Yaskawa INFORM job: ARGAZ5.JBI

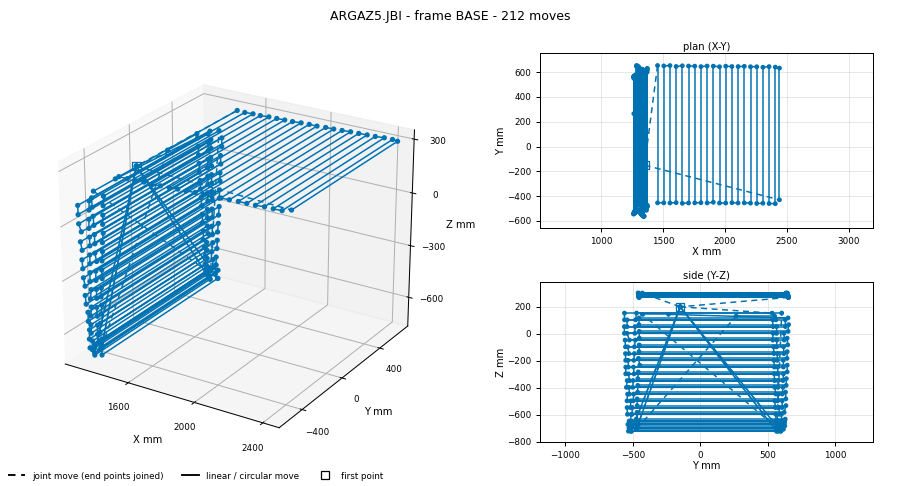
[picture p0: tool path of ARGAZ5.JBI in frame BASE, 212 of 212 moves have a stored position in this frame; points joined in program order, loops and branches not executed]
/JOB
//NAME ARGAZ5
//POS
///NPOS 206,0,206,1,0,1
///TOOL 0
///POSTYPE BASE
///RECTAN
///RCONF 0,0,0,0,0,0,0,0,0,0,0,0,0,0,0,0,0,0,0,0,0,0,0,0
C00000=2438.372,-429.843,302.316,175.0000,5.0000,175.0000
C00001=2438.372,633.343,302.316,175.0000,5.0000,175.0000
C00002=2404.704,640.901,302.803,175.0000,5.0000,175.0000
C00003=2404.704,-461.113,302.803,175.0000,5.0000,175.0000
C00004=2354.704,-459.538,300.563,175.0000,5.0000,175.0000
C00005=2354.704,645.007,300.563,175.0000,5.0000,175.0000
C00006=2304.704,639.966,299.253,175.0000,5.0000,175.0000
C00007=2304.704,-457.215,299.253,175.0000,5.0000,175.0000
C00008=2254.704,-459.172,296.365,175.0000,5.0000,175.0000
C00009=2254.704,644.031,296.365,175.0000,5.0000,175.0000
C00010=2204.704,644.248,294.144,175.0000,5.0000,175.0000
C00011=2204.704,-456.654,294.144,175.0000,5.0000,175.0000
C00012=2154.704,-454.150,292.149,175.0000,5.0000,175.0000
C00013=2154.704,647.282,292.149,175.0000,5.0000,175.0000
C00014=2104.704,645.426,290.068,175.0000,5.0000,175.0000
C00015=2104.704,-455.328,290.068,175.0000,5.0000,175.0000
C00016=2054.704,-453.054,287.793,175.0000,5.0000,175.0000
C00017=2054.704,645.839,287.793,175.0000,5.0000,175.0000
C00018=2004.704,648.293,285.625,175.0000,5.0000,175.0000
C00019=2004.704,-455.974,285.625,175.0000,5.0000,175.0000
C00020=1954.704,-455.663,284.513,175.0000,5.0000,175.0000
C00021=1954.704,644.044,284.513,175.0000,5.0000,175.0000
C00022=1904.704,648.760,282.533,175.0000,5.0000,175.0000
C00023=1904.704,-449.454,282.533,175.0000,5.0000,175.0000
C00024=1854.704,-454.861,280.617,175.0000,5.0000,175.0000
C00025=1854.704,649.609,280.617,175.0000,5.0000,175.0000
C00026=1804.704,645.165,279.272,175.0000,5.0000,175.0000
C00027=1804.704,-453.058,279.272,175.0000,5.0000,175.0000
C00028=1754.704,-454.350,276.998,175.0000,5.0000,175.0000
C00029=1754.704,648.797,276.998,175.0000,5.0000,175.0000
C00030=1704.704,649.851,275.425,175.0000,5.0000,175.0000
C00031=1704.704,-455.236,275.425,175.0000,5.0000,175.0000
C00032=1654.704,-457.856,273.661,175.0000,5.0000,175.0000
C00033=1654.704,651.982,273.661,175.0000,5.0000,175.0000
C00034=1604.704,646.210,272.661,175.0000,5.0000,175.0000
C00035=1604.704,-452.258,272.661,175.0000,5.0000,175.0000
C00036=1554.704,-455.193,270.474,175.0000,5.0000,175.0000
C00037=1554.704,653.496,270.474,175.0000,5.0000,175.0000
C00038=1504.704,650.879,269.338,175.0000,5.0000,175.0000
C00039=1504.704,-454.045,269.338,175.0000,5.0000,175.0000
C00040=1454.676,-454.040,269.843,175.0000,5.0000,175.0000
C00041=1454.676,653.895,269.843,175.0000,5.0000,175.0000
C00042=1347.088,531.287,153.366,175.0000,-89.9999,5.0000
C00043=1347.088,-562.394,153.366,175.0000,-89.9999,5.0000
C00044=1344.164,-562.287,103.366,175.0000,-89.9999,5.0000
C00045=1344.164,534.938,103.366,175.0000,-89.9999,5.0000
C00046=1342.438,538.625,53.366,175.0000,-89.9999,5.0000
C00047=1342.438,-562.994,53.366,175.0000,-89.9999,5.0000
C00048=1340.832,-563.178,3.366,175.0000,-89.9999,5.0000
C00049=1340.832,538.871,3.366,175.0000,-89.9999,5.0000
C00050=1338.825,536.219,-46.633,175.0000,-89.9999,5.0000
C00051=1338.825,-558.107,-46.633,175.0000,-89.9999,5.0000
C00052=1337.044,-554.870,-96.633,175.0000,-89.9999,5.0000
C00053=1337.044,542.164,-96.633,175.0000,-89.9999,5.0000
C00054=1335.183,545.111,-146.633,175.0000,-89.9999,5.0000
C00055=1335.183,-555.018,-146.633,175.0000,-89.9999,5.0000
C00056=1333.293,-553.493,-196.633,175.0000,-89.9999,5.0000
C00057=1333.293,545.184,-196.633,175.0000,-89.9999,5.0000
C00058=1331.807,548.689,-246.633,175.0000,-89.9999,5.0000
C00059=1331.807,-552.923,-246.633,175.0000,-89.9999,5.0000
C00060=1329.870,-553.256,-296.633,175.0000,-89.9999,5.0000
C00061=1329.870,547.209,-296.633,175.0000,-89.9999,5.0000
C00062=1327.995,549.873,-346.633,175.0000,-89.9999,5.0000
C00063=1327.995,-542.334,-346.633,175.0000,-89.9999,5.0000
C00064=1326.213,-548.248,-396.633,175.0000,-89.9999,5.0000
C00065=1326.213,550.626,-396.633,175.0000,-89.9999,5.0000
C00066=1324.396,560.131,-446.633,175.0000,-89.9999,5.0000
C00067=1324.396,-539.231,-446.633,175.0000,-89.9999,5.0000
C00068=1322.129,-543.451,-496.633,175.0000,-89.9999,5.0000
C00069=1322.129,550.722,-496.633,175.0000,-89.9999,5.0000
C00070=1320.170,556.350,-546.633,175.0000,-89.9999,5.0000
C00071=1320.170,-543.270,-546.633,175.0000,-89.9999,5.0000
C00072=1318.250,-540.170,-596.633,175.0000,-89.9999,5.0000
C00073=1318.250,558.973,-596.633,175.0000,-89.9999,5.0000
C00074=1316.642,560.301,-646.633,175.0000,-89.9999,5.0000
C00075=1316.642,-527.964,-646.633,175.0000,-89.9999,5.0000
C00076=1314.806,-529.352,-696.633,175.0000,-89.9999,5.0000
C00077=1314.806,561.085,-696.633,175.0000,-89.9999,5.0000
C00078=1333.412,565.195,-671.633,180.0000,-60.0000,0.0000
C00079=1333.412,-537.251,-671.633,180.0000,-60.0000,0.0000
C00080=1332.156,-533.079,-721.633,180.0000,-60.0000,0.0000
C00081=1332.156,565.345,-721.633,180.0000,-60.0000,0.0000
C00082=1332.156,565.345,-721.633,180.0000,-60.0000,0.0000
C00083=1371.377,602.641,153.649,175.0000,-89.9999,5.0000
C00084=1371.377,-472.613,153.649,175.0000,-89.9999,5.0000
C00085=1372.180,-480.408,103.649,175.0000,-89.9999,5.0000
C00086=1372.180,629.123,103.649,175.0000,-89.9999,5.0000
C00087=1371.089,629.796,53.649,175.0000,-89.9999,5.0000
C00088=1371.089,-483.667,53.649,175.0000,-89.9999,5.0000
C00089=1369.998,-485.573,3.649,175.0000,-89.9999,5.0000
C00090=1369.998,619.394,3.649,175.0000,-89.9999,5.0000
C00091=1369.110,621.830,-46.350,175.0000,-89.9999,5.0000
C00092=1369.110,-481.873,-46.350,175.0000,-89.9999,5.0000
C00093=1367.639,-488.976,-96.350,175.0000,-89.9999,5.0000
C00094=1367.639,616.630,-96.350,175.0000,-89.9999,5.0000
C00095=1366.582,618.500,-146.350,175.0000,-89.9999,5.0000
C00096=1366.582,-488.746,-146.350,175.0000,-89.9999,5.0000
C00097=1365.085,-493.213,-196.350,175.0000,-89.9999,5.0000
C00098=1365.085,614.650,-196.350,175.0000,-89.9999,5.0000
C00099=1363.658,614.990,-246.350,175.0000,-89.9999,5.0000
C00100=1363.658,-495.754,-246.350,175.0000,-89.9999,5.0000
C00101=1361.864,-491.909,-296.350,175.0000,-89.9999,5.0000
C00102=1361.864,615.571,-296.350,175.0000,-89.9999,5.0000
C00103=1360.073,611.872,-346.350,175.0000,-89.9999,5.0000
C00104=1360.073,-498.655,-346.350,175.0000,-89.9999,5.0000
C00105=1358.161,-500.748,-396.350,175.0000,-89.9999,5.0000
C00106=1358.161,611.928,-396.350,175.0000,-89.9999,5.0000
C00107=1356.405,607.009,-446.350,175.0000,-89.9999,5.0000
C00108=1356.405,-493.709,-446.350,175.0000,-89.9999,5.0000
C00109=1354.608,-498.341,-496.350,175.0000,-89.9999,5.0000
C00110=1354.608,606.376,-496.350,175.0000,-89.9999,5.0000
C00111=1352.468,605.807,-546.350,175.0000,-89.9999,5.0000
C00112=1352.468,-503.981,-546.350,175.0000,-89.9999,5.0000
C00113=1350.405,-507.600,-596.350,175.0000,-89.9999,5.0000
C00114=1350.405,600.519,-596.350,175.0000,-89.9999,5.0000
C00115=1348.479,602.258,-646.350,175.0000,-89.9999,5.0000
C00116=1348.479,-507.412,-646.350,175.0000,-89.9999,5.0000
C00117=1346.462,-509.588,-696.350,175.0000,-89.9999,5.0000
C00118=1346.462,597.739,-696.350,175.0000,-89.9999,5.0000
C00119=1364.869,596.218,-671.350,180.0000,-60.0000,0.0000
C00120=1364.869,-512.867,-671.350,180.0000,-60.0000,0.0000
C00121=1363.104,-512.908,-721.350,180.0000,-60.0000,0.0000
C00122=1363.104,596.344,-721.350,180.0000,-60.0000,0.0000
C00123=1363.104,596.344,-721.350,180.0000,-60.0000,0.0000
C00124=1277.888,-429.618,144.199,175.0000,-89.9999,5.0000
C00125=1277.888,-236.558,144.199,175.0000,-89.9999,5.0000
C00126=1283.410,649.398,117.816,175.0000,-89.9999,5.0000
C00127=1283.410,-454.812,117.816,175.0000,-89.9999,5.0000
C00128=1286.253,-455.480,67.816,175.0000,-89.9999,5.0000
C00129=1286.253,653.737,67.816,175.0000,-89.9999,5.0000
C00130=1288.733,650.101,17.816,175.0000,-89.9999,5.0000
C00131=1288.733,-453.231,17.816,175.0000,-89.9999,5.0000
C00132=1291.050,-452.345,-32.183,175.0000,-89.9999,5.0000
C00133=1291.050,643.233,-32.183,175.0000,-89.9999,5.0000
C00134=1293.592,647.319,-82.183,175.0000,-89.9999,5.0000
C00135=1293.592,-453.386,-82.183,175.0000,-89.9999,5.0000
C00136=1295.614,-454.881,-132.183,175.0000,-89.9999,5.0000
C00137=1295.614,643.520,-132.183,175.0000,-89.9999,5.0000
C00138=1297.247,642.008,-182.183,175.0000,-89.9999,5.0000
C00139=1297.247,-459.228,-182.183,175.0000,-89.9999,5.0000
C00140=1299.433,-449.216,-232.183,175.0000,-89.9999,5.0000
C00141=1299.433,643.471,-232.183,175.0000,-89.9999,5.0000
C00142=1300.418,643.420,-282.183,175.0000,-89.9999,5.0000
C00143=1300.418,-460.256,-282.183,175.0000,-89.9999,5.0000
C00144=1302.234,-463.734,-332.183,175.0000,-89.9999,5.0000
C00145=1302.234,636.925,-332.183,175.0000,-89.9999,5.0000
C00146=1303.707,635.868,-382.183,175.0000,-89.9999,5.0000
C00147=1303.707,-463.869,-382.183,175.0000,-89.9999,5.0000
C00148=1305.086,-465.019,-432.183,175.0000,-89.9999,5.0000
C00149=1305.086,630.756,-432.183,175.0000,-89.9999,5.0000
C00150=1306.071,633.429,-482.183,175.0000,-89.9999,5.0000
C00151=1306.071,-468.802,-482.183,175.0000,-89.9999,5.0000
C00152=1307.412,-468.117,-532.183,175.0000,-89.9999,5.0000
C00153=1307.412,633.875,-532.183,175.0000,-89.9999,5.0000
C00154=1308.466,621.089,-582.183,175.0000,-89.9999,5.0000
C00155=1308.466,-469.996,-582.183,175.0000,-89.9999,5.0000
C00156=1310.304,-475.204,-632.183,175.0000,-89.9999,5.0000
C00157=1310.304,628.888,-632.183,175.0000,-89.9999,5.0000
C00158=1311.312,625.813,-682.183,175.0000,-89.9999,5.0000
C00159=1311.312,-473.494,-682.183,175.0000,-89.9999,5.0000
C00160=1332.658,-465.818,-657.183,180.0000,-60.0000,0.0000
C00161=1332.658,624.168,-657.183,180.0000,-60.0000,0.0000
C00162=1333.118,615.110,-707.183,180.0000,-60.0000,0.0000
C00163=1333.118,-474.618,-707.183,180.0000,-60.0000,0.0000
C00164=1333.118,-474.618,-707.183,180.0000,-60.0000,0.0000
C00165=1263.288,265.502,131.277,175.0000,-89.9999,5.0000
C00166=1263.288,550.035,131.277,175.0000,-89.9999,5.0000
C00167=1260.890,559.755,103.296,175.0000,-89.9999,5.0000
C00168=1260.890,-543.266,103.296,175.0000,-89.9999,5.0000
C00169=1261.533,-543.209,53.296,175.0000,-89.9999,5.0000
C00170=1261.533,565.502,53.296,175.0000,-89.9999,5.0000
C00171=1263.366,564.257,3.296,175.0000,-89.9999,5.0000
C00172=1263.366,-543.096,3.296,175.0000,-89.9999,5.0000
C00173=1265.404,-525.948,-46.703,175.0000,-89.9999,5.0000
C00174=1265.404,566.502,-46.703,175.0000,-89.9999,5.0000
C00175=1267.028,564.815,-96.703,175.0000,-89.9999,5.0000
C00176=1267.028,-538.386,-96.703,175.0000,-89.9999,5.0000
C00177=1269.183,-528.977,-146.703,175.0000,-89.9999,5.0000
C00178=1269.183,570.662,-146.703,175.0000,-89.9999,5.0000
C00179=1270.966,569.787,-196.703,175.0000,-89.9999,5.0000
C00180=1270.966,-535.503,-196.703,175.0000,-89.9999,5.0000
C00181=1272.925,-533.396,-246.703,175.0000,-89.9999,5.0000
C00182=1272.925,572.645,-246.703,175.0000,-89.9999,5.0000
C00183=1275.047,573.565,-296.703,175.0000,-89.9999,5.0000
C00184=1275.047,-533.499,-296.703,175.0000,-89.9999,5.0000
C00185=1277.369,-524.427,-346.703,175.0000,-89.9999,5.0000
C00186=1277.369,576.345,-346.703,175.0000,-89.9999,5.0000
C00187=1279.521,573.757,-396.703,175.0000,-89.9999,5.0000
C00188=1279.521,-528.930,-396.703,175.0000,-89.9999,5.0000
C00189=1281.635,-525.764,-446.703,175.0000,-89.9999,5.0000
C00190=1281.635,579.175,-446.703,175.0000,-89.9999,5.0000
C00191=1283.849,571.736,-496.703,175.0000,-89.9999,5.0000
C00192=1283.849,-515.793,-496.703,175.0000,-89.9999,5.0000
C00193=1285.977,-517.912,-546.703,175.0000,-89.9999,5.0000
C00194=1285.977,582.744,-546.703,175.0000,-89.9999,5.0000
C00195=1288.303,585.349,-596.703,175.0000,-89.9999,5.0000
C00196=1288.303,-512.618,-596.703,175.0000,-89.9999,5.0000
C00197=1290.270,-519.107,-646.703,175.0000,-89.9999,5.0000
C00198=1290.270,579.567,-646.703,175.0000,-89.9999,5.0000
C00199=1292.656,581.655,-696.703,175.0000,-89.9999,5.0000
C00200=1292.656,-518.761,-696.703,175.0000,-89.9999,5.0000
C00201=1314.870,-511.376,-671.703,180.0000,-60.0000,0.0000
C00202=1314.870,581.349,-671.703,180.0000,-60.0000,0.0000
C00203=1317.105,581.261,-721.703,180.0000,-60.0000,0.0000
C00204=1317.105,-511.969,-721.703,180.0000,-60.0000,0.0000
C00205=1317.105,-511.969,-721.703,180.0000,-60.0000,0.0000
///POSTYPE PULSE
///PULSE
EC00000=0
EC00001=0
EC00002=0
EC00003=0
EC00004=0
EC00005=0
EC00006=0
EC00007=0
EC00008=0
EC00009=0
EC00010=0
EC00011=0
EC00012=0
EC00013=0
EC00014=0
EC00015=0
EC00016=0
EC00017=0
EC00018=0
EC00019=0
EC00020=0
EC00021=0
EC00022=0
EC00023=0
EC00024=0
EC00025=0
EC00026=0
EC00027=0
EC00028=0
EC00029=0
EC00030=0
EC00031=0
EC00032=0
EC00033=0
EC00034=0
EC00035=0
EC00036=0
EC00037=0
EC00038=0
EC00039=0
EC00040=0
EC00041=0
EC00042=0
EC00043=0
EC00044=0
EC00045=0
EC00046=0
EC00047=0
EC00048=0
EC00049=0
EC00050=0
EC00051=0
EC00052=0
EC00053=0
EC00054=0
EC00055=0
EC00056=0
EC00057=0
EC00058=0
EC00059=0
EC00060=0
EC00061=0
EC00062=0
EC00063=0
EC00064=0
EC00065=0
EC00066=0
EC00067=0
EC00068=0
EC00069=0
EC00070=0
EC00071=0
EC00072=0
EC00073=0
EC00074=0
EC00075=0
EC00076=0
EC00077=0
EC00078=0
EC00079=0
EC00080=0
EC00081=0
EC00082=92160
EC00083=92160
EC00084=92160
EC00085=92160
EC00086=92160
EC00087=92160
EC00088=92160
EC00089=92160
EC00090=92160
EC00091=92160
EC00092=92160
EC00093=92160
EC00094=92160
EC00095=92160
EC00096=92160
EC00097=92160
EC00098=92160
EC00099=92160
EC00100=92160
EC00101=92160
EC00102=92160
EC00103=92160
EC00104=92160
EC00105=92160
EC00106=92160
EC00107=92160
EC00108=92160
EC00109=92160
EC00110=92160
EC00111=92160
EC00112=92160
EC00113=92160
EC00114=92160
EC00115=92160
EC00116=92160
EC00117=92160
EC00118=92160
EC00119=92160
EC00120=92160
EC00121=92160
EC00122=92160
EC00123=184320
EC00124=184320
EC00125=184320
EC00126=184320
EC00127=184320
EC00128=184320
EC00129=184320
EC00130=184320
EC00131=184320
EC00132=184320
EC00133=184320
EC00134=184320
EC00135=184320
EC00136=184320
EC00137=184320
EC00138=184320
EC00139=184320
EC00140=184320
EC00141=184320
EC00142=184320
EC00143=184320
EC00144=184320
EC00145=184320
EC00146=184320
EC00147=184320
EC00148=184320
EC00149=184320
EC00150=184320
EC00151=184320
EC00152=184320
EC00153=184320
EC00154=184320
EC00155=184320
EC00156=184320
EC00157=184320
EC00158=184320
EC00159=184320
EC00160=184320
EC00161=184320
EC00162=184320
EC00163=184320
EC00164=276480
EC00165=276480
EC00166=276480
EC00167=276480
EC00168=276480
EC00169=276480
EC00170=276480
EC00171=276480
EC00172=276480
EC00173=276480
EC00174=276480
EC00175=276480
EC00176=276480
EC00177=276480
EC00178=276480
EC00179=276480
EC00180=276480
EC00181=276480
EC00182=276480
EC00183=276480
EC00184=276480
EC00185=276480
EC00186=276480
EC00187=276480
EC00188=276480
EC00189=276480
EC00190=276480
EC00191=276480
EC00192=276480
EC00193=276480
EC00194=276480
EC00195=276480
EC00196=276480
EC00197=276480
EC00198=276480
EC00199=276480
EC00200=276480
EC00201=276480
EC00202=276480
EC00203=276480
EC00204=276480
EC00205=368640
///POSTYPE BASE
///RECTAN
///RCONF 1,0,0,0,0,0,0,0,0,0,0,0,0,0,0,0,0,0,0,0,0,0,0,0
P00009=1350.000,-150.000,200.000,-180.0000,-45.0000,0.0000
///POSTYPE PULSE
///PULSE
EX00000=0
//INST
///DATE 2023/01/29 16:16
///ATTR SC,RW,RJ
////FRAME BASE
///GROUP1 RB1,ST1
NOP
MOVJ P009 EX000 VJ=15.00
MOVJ C00000 EC00000 VJ=15.00
CALL JOB:SPYON
MOVL C00001 EC00001 V=150.0
MOVL C00002 EC00002 V=150.0
MOVL C00003 EC00003 V=150.0
MOVL C00004 EC00004 V=150.0
MOVL C00005 EC00005 V=150.0
MOVL C00006 EC00006 V=150.0
MOVL C00007 EC00007 V=150.0
MOVL C00008 EC00008 V=150.0
MOVL C00009 EC00009 V=150.0
MOVL C00010 EC00010 V=150.0
MOVL C00011 EC00011 V=150.0
MOVL C00012 EC00012 V=150.0
MOVL C00013 EC00013 V=150.0
MOVL C00014 EC00014 V=150.0
MOVL C00015 EC00015 V=150.0
MOVL C00016 EC00016 V=150.0
MOVL C00017 EC00017 V=150.0
MOVL C00018 EC00018 V=150.0
MOVL C00019 EC00019 V=150.0
MOVL C00020 EC00020 V=150.0
MOVL C00021 EC00021 V=150.0
MOVL C00022 EC00022 V=150.0
MOVL C00023 EC00023 V=150.0
MOVL C00024 EC00024 V=150.0
MOVL C00025 EC00025 V=150.0
MOVL C00026 EC00026 V=150.0
MOVL C00027 EC00027 V=150.0
MOVL C00028 EC00028 V=150.0
MOVL C00029 EC00029 V=150.0
MOVL C00030 EC00030 V=150.0
MOVL C00031 EC00031 V=150.0
MOVL C00032 EC00032 V=150.0
MOVL C00033 EC00033 V=150.0
MOVL C00034 EC00034 V=150.0
MOVL C00035 EC00035 V=150.0
MOVL C00036 EC00036 V=150.0
MOVL C00037 EC00037 V=150.0
MOVL C00038 EC00038 V=150.0
MOVL C00039 EC00039 V=150.0
MOVL C00040 EC00040 V=150.0
MOVL C00041 EC00041 V=150.0
CALL JOB:SPYOF
MOVJ P009 VJ=15.00
MOVJ C00042 EC00042 VJ=15.00
CALL JOB:SPYON
MOVL C00043 EC00043 V=150.0
MOVL C00044 EC00044 V=150.0
MOVL C00045 EC00045 V=150.0
MOVL C00046 EC00046 V=150.0
MOVL C00047 EC00047 V=150.0
MOVL C00048 EC00048 V=150.0
MOVL C00049 EC00049 V=150.0
MOVL C00050 EC00050 V=150.0
MOVL C00051 EC00051 V=150.0
MOVL C00052 EC00052 V=150.0
MOVL C00053 EC00053 V=150.0
MOVL C00054 EC00054 V=150.0
MOVL C00055 EC00055 V=150.0
MOVL C00056 EC00056 V=150.0
MOVL C00057 EC00057 V=150.0
MOVL C00058 EC00058 V=150.0
MOVL C00059 EC00059 V=150.0
MOVL C00060 EC00060 V=150.0
MOVL C00061 EC00061 V=150.0
MOVL C00062 EC00062 V=150.0
MOVL C00063 EC00063 V=150.0
MOVL C00064 EC00064 V=150.0
MOVL C00065 EC00065 V=150.0
MOVL C00066 EC00066 V=150.0
MOVL C00067 EC00067 V=150.0
MOVL C00068 EC00068 V=150.0
MOVL C00069 EC00069 V=150.0
MOVL C00070 EC00070 V=150.0
MOVL C00071 EC00071 V=150.0
MOVL C00072 EC00072 V=150.0
MOVL C00073 EC00073 V=150.0
MOVL C00074 EC00074 V=150.0
MOVL C00075 EC00075 V=150.0
MOVL C00076 EC00076 V=150.0
MOVL C00077 EC00077 V=150.0
MOVL C00078 EC00078 V=150.0
MOVL C00079 EC00079 V=150.0
MOVL C00080 EC00080 V=150.0
MOVL C00081 EC00081 V=150.0
CALL JOB:SPYOF
MOVJ P009 VJ=15.00
MOVL C00082 EC00082 V=150.0
MOVJ C00083 EC00083 VJ=15.00
CALL JOB:SPYON
MOVL C00084 EC00084 V=150.0
MOVL C00085 EC00085 V=150.0
MOVL C00086 EC00086 V=150.0
MOVL C00087 EC00087 V=150.0
MOVL C00088 EC00088 V=150.0
MOVL C00089 EC00089 V=150.0
MOVL C00090 EC00090 V=150.0
MOVL C00091 EC00091 V=150.0
MOVL C00092 EC00092 V=150.0
MOVL C00093 EC00093 V=150.0
MOVL C00094 EC00094 V=150.0
MOVL C00095 EC00095 V=150.0
MOVL C00096 EC00096 V=150.0
MOVL C00097 EC00097 V=150.0
MOVL C00098 EC00098 V=150.0
MOVL C00099 EC00099 V=150.0
MOVL C00100 EC00100 V=150.0
MOVL C00101 EC00101 V=150.0
MOVL C00102 EC00102 V=150.0
MOVL C00103 EC00103 V=150.0
MOVL C00104 EC00104 V=150.0
MOVL C00105 EC00105 V=150.0
MOVL C00106 EC00106 V=150.0
MOVL C00107 EC00107 V=150.0
MOVL C00108 EC00108 V=150.0
MOVL C00109 EC00109 V=150.0
MOVL C00110 EC00110 V=150.0
MOVL C00111 EC00111 V=150.0
MOVL C00112 EC00112 V=150.0
MOVL C00113 EC00113 V=150.0
MOVL C00114 EC00114 V=150.0
MOVL C00115 EC00115 V=150.0
MOVL C00116 EC00116 V=150.0
MOVL C00117 EC00117 V=150.0
MOVL C00118 EC00118 V=150.0
MOVL C00119 EC00119 V=150.0
MOVL C00120 EC00120 V=150.0
MOVL C00121 EC00121 V=150.0
MOVL C00122 EC00122 V=150.0
CALL JOB:SPYOF
MOVJ P009 VJ=15.00
MOVL C00123 EC00123 V=150.0
MOVJ C00124 EC00124 VJ=15.00
CALL JOB:SPYON
MOVL C00125 EC00125 V=150.0
MOVL C00126 EC00126 V=150.0
MOVL C00127 EC00127 V=150.0
MOVL C00128 EC00128 V=150.0
MOVL C00129 EC00129 V=150.0
MOVL C00130 EC00130 V=150.0
MOVL C00131 EC00131 V=150.0
MOVL C00132 EC00132 V=150.0
MOVL C00133 EC00133 V=150.0
MOVL C00134 EC00134 V=150.0
MOVL C00135 EC00135 V=150.0
MOVL C00136 EC00136 V=150.0
MOVL C00137 EC00137 V=150.0
MOVL C00138 EC00138 V=150.0
MOVL C00139 EC00139 V=150.0
MOVL C00140 EC00140 V=150.0
MOVL C00141 EC00141 V=150.0
MOVL C00142 EC00142 V=150.0
MOVL C00143 EC00143 V=150.0
MOVL C00144 EC00144 V=150.0
MOVL C00145 EC00145 V=150.0
MOVL C00146 EC00146 V=150.0
MOVL C00147 EC00147 V=150.0
MOVL C00148 EC00148 V=150.0
MOVL C00149 EC00149 V=150.0
MOVL C00150 EC00150 V=150.0
MOVL C00151 EC00151 V=150.0
MOVL C00152 EC00152 V=150.0
MOVL C00153 EC00153 V=150.0
MOVL C00154 EC00154 V=150.0
MOVL C00155 EC00155 V=150.0
MOVL C00156 EC00156 V=150.0
MOVL C00157 EC00157 V=150.0
MOVL C00158 EC00158 V=150.0
MOVL C00159 EC00159 V=150.0
MOVL C00160 EC00160 V=150.0
MOVL C00161 EC00161 V=150.0
MOVL C00162 EC00162 V=150.0
MOVL C00163 EC00163 V=150.0
CALL JOB:SPYOF
MOVJ P009 VJ=15.00
MOVL C00164 EC00164 V=150.0
MOVJ C00165 EC00165 VJ=15.00
CALL JOB:SPYON
MOVL C00166 EC00166 V=150.0
MOVL C00167 EC00167 V=150.0
MOVL C00168 EC00168 V=150.0
MOVL C00169 EC00169 V=150.0
MOVL C00170 EC00170 V=150.0
MOVL C00171 EC00171 V=150.0
MOVL C00172 EC00172 V=150.0
MOVL C00173 EC00173 V=150.0
MOVL C00174 EC00174 V=150.0
MOVL C00175 EC00175 V=150.0
MOVL C00176 EC00176 V=150.0
MOVL C00177 EC00177 V=150.0
MOVL C00178 EC00178 V=150.0
MOVL C00179 EC00179 V=150.0
MOVL C00180 EC00180 V=150.0
MOVL C00181 EC00181 V=150.0
MOVL C00182 EC00182 V=150.0
MOVL C00183 EC00183 V=150.0
MOVL C00184 EC00184 V=150.0
MOVL C00185 EC00185 V=150.0
MOVL C00186 EC00186 V=150.0
MOVL C00187 EC00187 V=150.0
MOVL C00188 EC00188 V=150.0
MOVL C00189 EC00189 V=150.0
MOVL C00190 EC00190 V=150.0
MOVL C00191 EC00191 V=150.0
MOVL C00192 EC00192 V=150.0
MOVL C00193 EC00193 V=150.0
MOVL C00194 EC00194 V=150.0
MOVL C00195 EC00195 V=150.0
MOVL C00196 EC00196 V=150.0
MOVL C00197 EC00197 V=150.0
MOVL C00198 EC00198 V=150.0
MOVL C00199 EC00199 V=150.0
MOVL C00200 EC00200 V=150.0
MOVL C00201 EC00201 V=150.0
MOVL C00202 EC00202 V=150.0
MOVL C00203 EC00203 V=150.0
MOVL C00204 EC00204 V=150.0
CALL JOB:SPYOF
MOVJ P009 VJ=15.00
MOVL C00205 EC00205 V=150.0
END
